(* CoDeSys 2.3 project: PRJ_LAB_AUTO_MAX4_V2200.pro *)
(* Title: Exam project *)
(* Version: 0.1 *)
(* Author: Federico M. Rossi *)
(* Description: Small project to take the exam.
Relased under MIT license. *)
(* Libraries: System_V002200.lib 3.4.06 14:28:36, PacDriveLib_V002002.lib 6.2.06 18:39:46 *)

(* Task configuration *)
TASK SymVisrtualAct (PRIORITY := 31, INTERVAL := T#100ms);
	SYM_PRG();
END_TASK
TASK Main (PRIORITY := 31, INTERVAL := T#10ms);
	PLC_PRG();
END_TASK

(* Global variable list: Global_Variables *)
VAR_GLOBAL
	tmpBool:BOOL;
	tmpReal:REAL;
	tmpDINT:DINT;
	tmpString:STRING(30);
	tmpTime:TIME;


	P1:virtual_piston_df_t;
	P2:virtual_piston_sfd_t;

	TP_PACK:BOOL:=FALSE;

	(* Machine config *)
	c:config_machine_t;




END_VAR

(* Data type *)
TYPE config_homing_t :
STRUCT
	maxTravel:REAL;
	vel:REAL;
	acc:REAL;
END_STRUCT
END_TYPE

(* Data type *)
TYPE config_machine_t :
STRUCT
	tape:config_tape_t;
	mov1:config_mov_t;
	mov2:config_mov_t;
	p1:config_piston_t;
	p2:config_piston_t;
	home1:config_homing_t;
	home2:config_homing_t;
END_STRUCT
END_TYPE

(* Data type *)
TYPE config_mov_t :
STRUCT
	acc:REAL;
	vel:REAL;
	pos:REAL;
	startForwAtTapePos:REAL;
	startBackAtTapePos:REAL;
END_STRUCT
END_TYPE

(* Data type *)
TYPE config_piston_t :
STRUCT
	deactAtTapePos:REAL;
END_STRUCT
END_TYPE

(* Data type *)
TYPE config_tape_t :
STRUCT
	acc:REAL;
	vel:REAL;
	period:REAL;
	packTimeoutSec:TIME;
END_STRUCT
END_TYPE

(* Data type *)
TYPE virtual_piston_df_i_t :
STRUCT
	setEnable:BOOL;
	setStart:BOOL;
END_STRUCT
END_TYPE

(* Data type *)
TYPE virtual_piston_df_o_t :
STRUCT
	isActive:BOOL;
	isOut:BOOL;
	isIn:BOOL;
END_STRUCT
END_TYPE

(* Data type *)
TYPE virtual_piston_df_t :
STRUCT
	i:virtual_piston_df_i_t;
	o:virtual_piston_df_o_t;
END_STRUCT
END_TYPE

(* Data type *)
TYPE virtual_piston_sfd_i_t :
STRUCT
	setEnable:BOOL;
	setStart:BOOL;
END_STRUCT
END_TYPE

(* Data type *)
TYPE virtual_piston_sfd_o_t :
STRUCT
	isActive:BOOL;
	isIn:BOOL;
END_STRUCT
END_TYPE

(* Data type *)
TYPE virtual_piston_sfd_t :
STRUCT
	i:virtual_piston_sfd_i_t;
	o:virtual_piston_sfd_o_t;
END_STRUCT
END_TYPE

(* POU SYM_PRG, ST *)
PROGRAM SYM_PRG
VAR

END_VAR
(* Piston 1 *)
IF ( P1.i.setEnable) THEN
	P1.o.isActive:=TRUE;
	IF ( P1.i.setStart) THEN
		p1.o.isIn:=FALSE;
		p1.o.isOut:=TRUE;
	ELSE
		p1.o.isIn:=TRUE;
		p1.o.isOut:=FALSE;
	END_IF
ELSE
	P1.o.isActive:=FALSE;
	P1.o.isIn:=FALSE;
	P1.o.isOut:=FALSE;
END_IF

(* Piston 2 *)
IF ( P2.i.setEnable) THEN
	P2.o.isActive:=TRUE;
	IF ( P2.i.setStart) THEN
		p2.o.isIn:=FALSE;
	ELSE
		p2.o.isIn:=TRUE;
	END_IF
ELSE
	P2.o.isActive:=FALSE;
	P2.o.isIn:=FALSE;
END_IF
END_PROGRAM

(* POU PLC_PRG, SFC *)
PROGRAM PLC_PRG
VAR
	exception:BOOL:=FALSE;

	(* axisMgmt => StateMachine *)
	enableOk:BOOL:=FALSE;
	homingOk:BOOL:=FALSE;
	syncStopOk:BOOL:=FALSE;
	tapeTimedOut:BOOL:=FALSE;
	(* StateMachine => axisMgmt *)
	AxisMgmtRoutine:INT:=0;

	(* tape related vars *)
	tape_pos_off:REAL;
	tape_pos_rel:REAL;
	flag_tp_pack:BOOL:=FALSE;
	timerTape:TON;
	jog1:Jogging3;
	jog2:Jogging3;
	elf_tape:EndlessFeed3;
	htp1:PDL_FB_HomeTP ;
	htp2:PDL_FB_HomeTP ;
	flagProcessingPack:BOOL;

	sm:STATE_MACHINE;
	OpModeReq:INT:=0;
	OpModeTimer:TON;
	stepReady:BOOL:=FALSE;
END_VAR
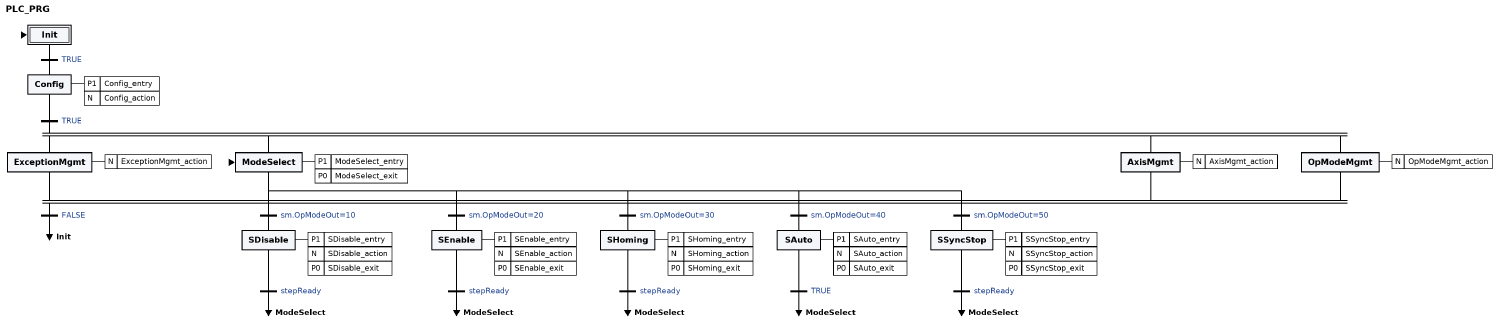
INITIAL_STEP Init:
END_STEP
TRANSITION FROM Init TO Config := TRUE;
END_TRANSITION
STEP Config:
	Config_entry(P1);
	Config_action(N);
END_STEP
TRANSITION FROM Config TO (ExceptionMgmt, ModeSelect, AxisMgmt, OpModeMgmt) := TRUE;
END_TRANSITION
STEP ExceptionMgmt:
	ExceptionMgmt_action(N);
END_STEP
STEP ModeSelect:
	ModeSelect_entry(P1);
	ModeSelect_exit(P0);
END_STEP
TRANSITION FROM ModeSelect TO SDisable := sm.OpModeOut=10;
END_TRANSITION
TRANSITION FROM ModeSelect TO SEnable := sm.OpModeOut=20;
END_TRANSITION
TRANSITION FROM ModeSelect TO SHoming := sm.OpModeOut=30;
END_TRANSITION
TRANSITION FROM ModeSelect TO SAuto := sm.OpModeOut=40;
END_TRANSITION
TRANSITION FROM ModeSelect TO SSyncStop := sm.OpModeOut=50;
END_TRANSITION
STEP SDisable:
	SDisable_entry(P1);
	SDisable_action(N);
	SDisable_exit(P0);
END_STEP
TRANSITION FROM SDisable TO ModeSelect := stepReady;
END_TRANSITION
STEP SEnable:
	SEnable_entry(P1);
	SEnable_action(N);
	SEnable_exit(P0);
END_STEP
TRANSITION FROM SEnable TO ModeSelect := stepReady;
END_TRANSITION
STEP SHoming:
	SHoming_entry(P1);
	SHoming_action(N);
	SHoming_exit(P0);
END_STEP
TRANSITION FROM SHoming TO ModeSelect := stepReady;
END_TRANSITION
STEP SAuto:
	SAuto_entry(P1);
	SAuto_action(N);
	SAuto_exit(P0);
END_STEP
TRANSITION FROM SAuto TO ModeSelect := TRUE;
END_TRANSITION
STEP SSyncStop:
	SSyncStop_entry(P1);
	SSyncStop_action(N);
	SSyncStop_exit(P0);
END_STEP
TRANSITION FROM SSyncStop TO ModeSelect := stepReady;
END_TRANSITION
STEP AxisMgmt:
	AxisMgmt_action(N);
END_STEP
STEP OpModeMgmt:
	OpModeMgmt_action(N);
END_STEP
TRANSITION FROM (ExceptionMgmt, AxisMgmt, OpModeMgmt) TO Init := FALSE;
END_TRANSITION

ACTION Config_entry:
	c.mov1.acc:=5000;
	c.mov1.pos:=90;
	c.mov1.startForwAtTapePos:=0;
	c.mov1.startBackAtTapePos:=180;
	c.mov1.vel:=90;

	c.mov2.acc:=5000;
	c.mov2.pos:=180;
	c.mov2.startForwAtTapePos:=360;
	c.mov2.startBackAtTapePos:=360+180;
	c.mov2.vel:=180;

	c.p1.deactAtTapePos:=180+45;
	c.p2.deactAtTapePos:=360+180+45;

	c.tape.acc:=5000;
	c.tape.packTimeoutSec:=t#30s;
	c.tape.period:=720;
	c.tape.vel:=72;

	c.home1.acc:=5000;
	c.home1.maxTravel:=750;
	c.home1.vel:=90;

	c.home2.acc:=5000;
	c.home2.maxTravel:=750;
	c.home2.vel:=90;
END_ACTION

ACTION Config_action:
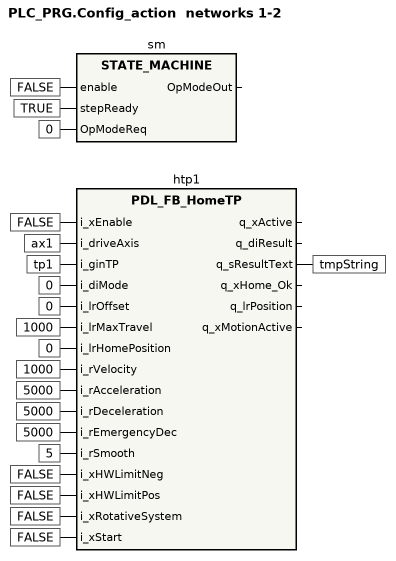
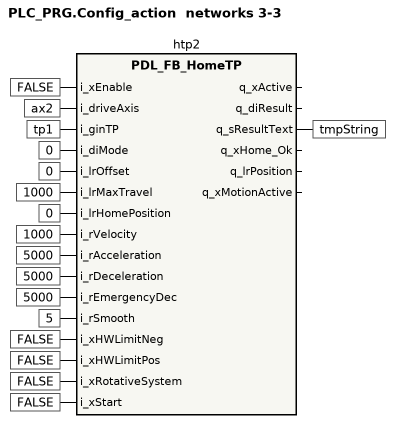
_FBD_ (* Function Block Diagram *)
NETWORK 1
	sm:STATE_MACHINE(enable: FALSE, stepReady: TRUE, OpModeReq: 0)
NETWORK 2
	htp1:PDL_FB_HomeTP(i_xEnable: FALSE, i_driveAxis: ax1, i_ginTP: tp1, i_diMode: 0, i_lrOffset: 0, i_lrMaxTravel: 1000, i_lrHomePosition: 0, i_rVelocity: 1000, i_rAcceleration: 5000, i_rDeceleration: 5000, i_rEmergencyDec: 5000, i_rSmooth: 5, i_xHWLimitNeg: FALSE, i_xHWLimitPos: FALSE, i_xRotativeSystem: FALSE, i_xStart: FALSE, q_sResultText => tmpString)
NETWORK 3
	htp2:PDL_FB_HomeTP(i_xEnable: FALSE, i_driveAxis: ax2, i_ginTP: tp1, i_diMode: 0, i_lrOffset: 0, i_lrMaxTravel: 1000, i_lrHomePosition: 0, i_rVelocity: 1000, i_rAcceleration: 5000, i_rDeceleration: 5000, i_rEmergencyDec: 5000, i_rSmooth: 5, i_xHWLimitNeg: FALSE, i_xHWLimitPos: FALSE, i_xRotativeSystem: FALSE, i_xStart: FALSE, q_sResultText => tmpString)
_END_FBD_
(* the same logic as Structured Text *)
(* Network 1 *)
sm(enable := FALSE, stepReady := TRUE, OpModeReq := 0);
(* Network 2 *)
htp1(i_xEnable := FALSE, i_driveAxis := ax1, i_ginTP := tp1, i_diMode := 0, i_lrOffset := 0, i_lrMaxTravel := 1000, i_lrHomePosition := 0, i_rVelocity := 1000, i_rAcceleration := 5000, i_rDeceleration := 5000, i_rEmergencyDec := 5000, i_rSmooth := 5, i_xHWLimitNeg := FALSE, i_xHWLimitPos := FALSE, i_xRotativeSystem := FALSE, i_xStart := FALSE);
tmpString := htp1.q_sResultText;
(* Network 3 *)
htp2(i_xEnable := FALSE, i_driveAxis := ax2, i_ginTP := tp1, i_diMode := 0, i_lrOffset := 0, i_lrMaxTravel := 1000, i_lrHomePosition := 0, i_rVelocity := 1000, i_rAcceleration := 5000, i_rDeceleration := 5000, i_rEmergencyDec := 5000, i_rSmooth := 5, i_xHWLimitNeg := FALSE, i_xHWLimitPos := FALSE, i_xRotativeSystem := FALSE, i_xStart := FALSE);
tmpString := htp2.q_sResultText;
END_ACTION

ACTION ExceptionMgmt_action:
(*
IF ( OpModeTimer.Q ) THEN
	exception:=TRUE;
END_IF
*)
IF (  exception ) THEN
	AxisMgmtRoutine:=0;
	stepReady:=TRUE;
	ax1.ControllerEnableSet:=FALSE;
	ax2.ControllerEnableSet:=FALSE;
	htp1.i_xEnable:=FALSE;
	htp2.i_xEnable:=FALSE;
	elf_tape.Enable:=FALSE;
	sm.enable:=FALSE;
END_IF
END_ACTION

ACTION ModeSelect_entry:
OpModeTimer.IN:=FALSE;
OpModeTimer.PT:=t#100s;
END_ACTION

ACTION ModeSelect_exit:
stepReady:=FALSE;
END_ACTION

ACTION SDisable_entry:
AxisMgmtRoutine:=10;
END_ACTION

ACTION SDisable_action:
IF ( (NOT enableOk) OR sm.OpModeOut<>10 ) THEN
	stepReady:=TRUE;
END_IF
END_ACTION

ACTION SDisable_exit:
AxisMgmtRoutine:=0;
END_ACTION

ACTION SEnable_entry:
AxisMgmtRoutine:=20;
OpModeTimer.PT:=t#10s;
OpModeTimer.IN:=TRUE;
END_ACTION

ACTION SEnable_action:
IF ( enableOk ) THEN
	stepReady:=TRUE;
END_IF
END_ACTION

ACTION SEnable_exit:
AxisMgmtRoutine:=0;
END_ACTION

ACTION SHoming_entry:
AxisMgmtRoutine:=30;
OpModeTimer.PT:=t#20s;
OpModeTimer.IN:=TRUE;
END_ACTION

ACTION SHoming_action:
IF ( homingOk ) THEN
	stepReady:=TRUE;
END_IF
END_ACTION

ACTION SHoming_exit:
AxisMgmtRoutine:=0;
END_ACTION

ACTION SAuto_entry:
OpModeTimer.IN:=FALSE;
END_ACTION

ACTION SAuto_action:
AxisMgmtRoutine:=40;
IF ( tapeTimedOut ) THEN
	OpModeReq:=50;
END_IF
END_ACTION

ACTION SAuto_exit:
AxisMgmtRoutine:=0;
END_ACTION

ACTION SSyncStop_entry:
OpModeTimer.IN:=FALSE;
END_ACTION

ACTION SSyncStop_action:
AxisMgmtRoutine:=50;
IF ( syncStopOk ) THEN
	stepReady:=TRUE;
END_IF
END_ACTION

ACTION SSyncStop_exit:
AxisMgmtRoutine:=0;
END_ACTION

ACTION AxisMgmt_action:
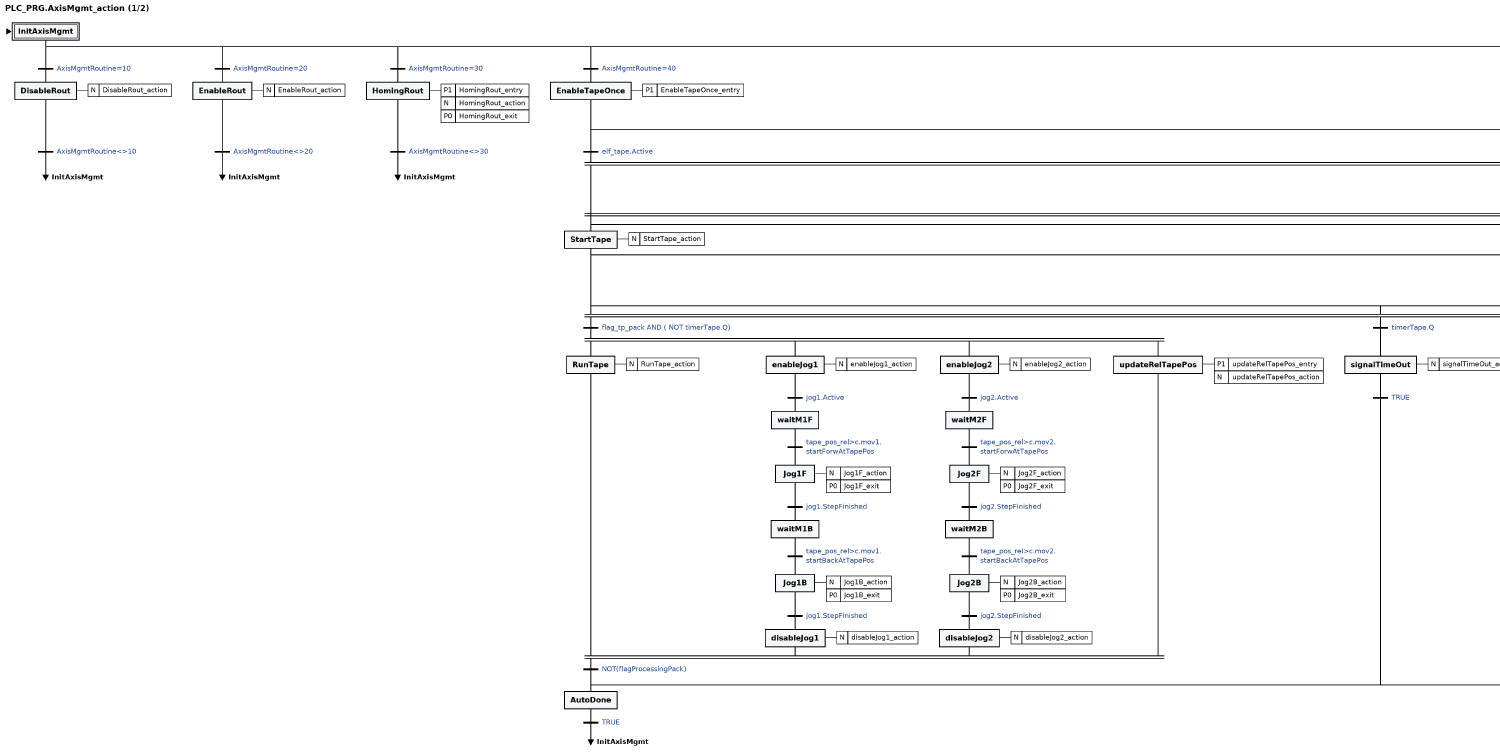
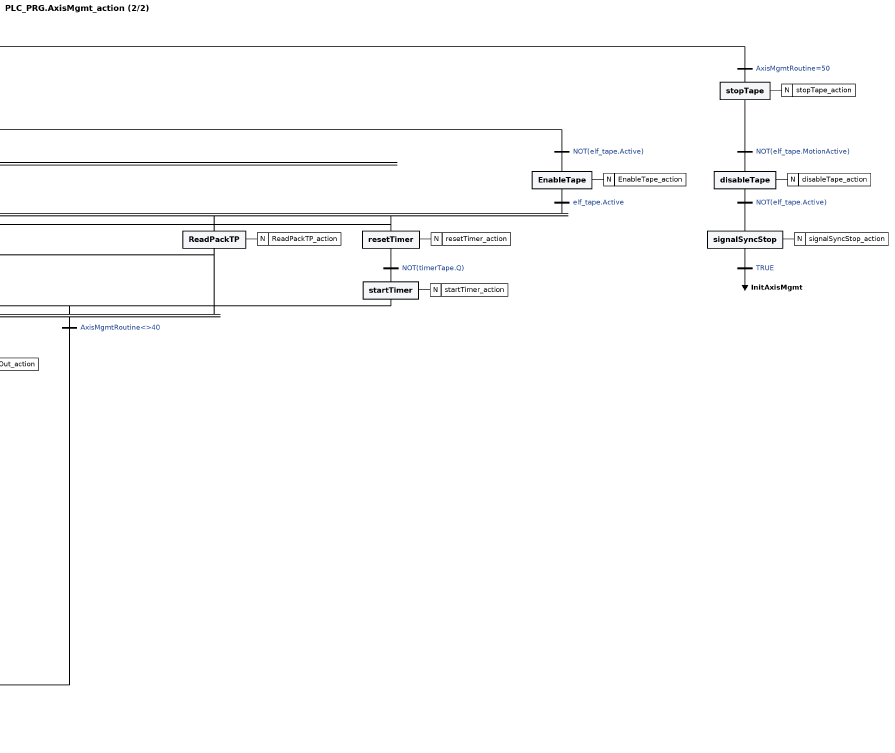
INITIAL_STEP InitAxisMgmt:
END_STEP
TRANSITION FROM InitAxisMgmt TO DisableRout := AxisMgmtRoutine=10;
END_TRANSITION
TRANSITION FROM InitAxisMgmt TO EnableRout := AxisMgmtRoutine=20;
END_TRANSITION
TRANSITION FROM InitAxisMgmt TO HomingRout := AxisMgmtRoutine=30;
END_TRANSITION
TRANSITION FROM InitAxisMgmt TO EnableTapeOnce := AxisMgmtRoutine=40;
END_TRANSITION
TRANSITION FROM InitAxisMgmt TO stopTape := AxisMgmtRoutine=50;
END_TRANSITION
STEP DisableRout:
	DisableRout_action(N);
END_STEP
TRANSITION FROM DisableRout TO InitAxisMgmt := AxisMgmtRoutine<>10;
END_TRANSITION
STEP EnableRout:
	EnableRout_action(N);
END_STEP
TRANSITION FROM EnableRout TO InitAxisMgmt := AxisMgmtRoutine<>20;
END_TRANSITION
STEP HomingRout:
	HomingRout_entry(P1);
	HomingRout_action(N);
	HomingRout_exit(P0);
END_STEP
TRANSITION FROM HomingRout TO InitAxisMgmt := AxisMgmtRoutine<>30;
END_TRANSITION
STEP EnableTapeOnce:
	EnableTapeOnce_entry(P1);
END_STEP
TRANSITION FROM EnableTapeOnce TO (StartTape, ReadPackTP, resetTimer) := elf_tape.Active;
END_TRANSITION
TRANSITION FROM EnableTapeOnce TO EnableTape := NOT(elf_tape.Active);
END_TRANSITION
STEP EnableTape:
	EnableTape_action(N);
END_STEP
TRANSITION FROM EnableTape TO (StartTape, ReadPackTP, resetTimer) := elf_tape.Active;
END_TRANSITION
STEP StartTape:
	StartTape_action(N);
END_STEP
STEP ReadPackTP:
	ReadPackTP_action(N);
END_STEP
STEP resetTimer:
	resetTimer_action(N);
END_STEP
TRANSITION FROM resetTimer TO startTimer := NOT(timerTape.Q);
END_TRANSITION
STEP startTimer:
	startTimer_action(N);
END_STEP
TRANSITION FROM (StartTape, ReadPackTP, startTimer) TO (RunTape, enableJog1, enableJog2, updateRelTapePos) := flag_tp_pack AND ( NOT timerTape.Q);
END_TRANSITION
TRANSITION FROM (StartTape, ReadPackTP, startTimer) TO signalTimeOut := timerTape.Q;
END_TRANSITION
TRANSITION FROM (StartTape, ReadPackTP, startTimer) TO AutoDone := AxisMgmtRoutine<>40;
END_TRANSITION
STEP RunTape:
	RunTape_action(N);
END_STEP
STEP enableJog1:
	enableJog1_action(N);
END_STEP
TRANSITION FROM enableJog1 TO waitM1F := jog1.Active;
END_TRANSITION
STEP waitM1F:
END_STEP
TRANSITION FROM waitM1F TO Jog1F := tape_pos_rel>c.mov1.startForwAtTapePos;
END_TRANSITION
STEP Jog1F:
	Jog1F_action(N);
	Jog1F_exit(P0);
END_STEP
TRANSITION FROM Jog1F TO waitM1B := jog1.StepFinished;
END_TRANSITION
STEP waitM1B:
END_STEP
TRANSITION FROM waitM1B TO Jog1B := tape_pos_rel>c.mov1.startBackAtTapePos;
END_TRANSITION
STEP Jog1B:
	Jog1B_action(N);
	Jog1B_exit(P0);
END_STEP
TRANSITION FROM Jog1B TO disableJog1 := jog1.StepFinished;
END_TRANSITION
STEP disableJog1:
	disableJog1_action(N);
END_STEP
STEP enableJog2:
	enableJog2_action(N);
END_STEP
TRANSITION FROM enableJog2 TO waitM2F := jog2.Active;
END_TRANSITION
STEP waitM2F:
END_STEP
TRANSITION FROM waitM2F TO Jog2F := tape_pos_rel>c.mov2.startForwAtTapePos;
END_TRANSITION
STEP Jog2F:
	Jog2F_action(N);
	Jog2F_exit(P0);
END_STEP
TRANSITION FROM Jog2F TO waitM2B := jog2.StepFinished;
END_TRANSITION
STEP waitM2B:
END_STEP
TRANSITION FROM waitM2B TO Jog2B := tape_pos_rel>c.mov2.startBackAtTapePos;
END_TRANSITION
STEP Jog2B:
	Jog2B_action(N);
	Jog2B_exit(P0);
END_STEP
TRANSITION FROM Jog2B TO disableJog2 := jog2.StepFinished;
END_TRANSITION
STEP disableJog2:
	disableJog2_action(N);
END_STEP
STEP updateRelTapePos:
	updateRelTapePos_entry(P1);
	updateRelTapePos_action(N);
END_STEP
TRANSITION FROM (RunTape, disableJog1, disableJog2, updateRelTapePos) TO AutoDone := NOT(flagProcessingPack);
END_TRANSITION
STEP signalTimeOut:
	signalTimeOut_action(N);
END_STEP
TRANSITION FROM signalTimeOut TO AutoDone := TRUE;
END_TRANSITION
STEP AutoDone:
END_STEP
TRANSITION FROM AutoDone TO InitAxisMgmt := TRUE;
END_TRANSITION
STEP stopTape:
	stopTape_action(N);
END_STEP
TRANSITION FROM stopTape TO disableTape := NOT(elf_tape.MotionActive);
END_TRANSITION
STEP disableTape:
	disableTape_action(N);
END_STEP
TRANSITION FROM disableTape TO signalSyncStop := NOT(elf_tape.Active);
END_TRANSITION
STEP signalSyncStop:
	signalSyncStop_action(N);
END_STEP
TRANSITION FROM signalSyncStop TO InitAxisMgmt := TRUE;
END_TRANSITION

ACTION DisableRout_action:
ax1.ControllerEnableSet := FALSE;
ax2.ControllerEnableSet := FALSE;
tape.ControllerEnableSet := FALSE;

IF ( ax1.AxisState=1 AND ax2.AxisState=1  ) THEN
	enableOk:=FALSE;
	homingOk:=FALSE;
	syncStopOk:=FALSE;
END_IF
END_ACTION

ACTION EnableRout_action:
ax1.ControllerEnableSet := TRUE;
ax2.ControllerEnableSet := TRUE;
tape.ControllerEnableSet := TRUE;

IF ( ax1.AxisState=3 AND ax2.AxisState=3 AND tape.AxisState=3) THEN
	enableOk:=TRUE;
	homingOk:=FALSE;
	syncStopOk:=FALSE;
ELSIF ( ax1.AxisState=8 OR ax2.AxisState=8 OR tape.AxisState=8  ) THEN
	exception:=TRUE;
END_IF
END_ACTION

ACTION HomingRout_entry:
htp1.i_xEnable:=TRUE;
htp2.i_xEnable:=TRUE;
homingOk:=FALSE;
syncStopOk:=FALSE;
END_ACTION

ACTION HomingRout_action:
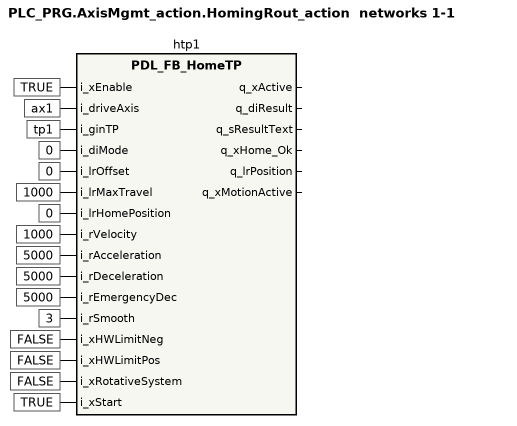
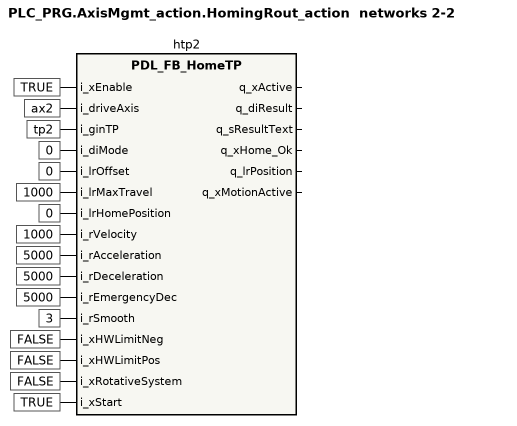
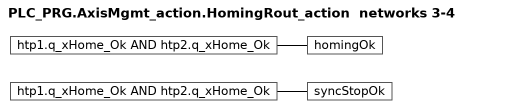
_FBD_ (* Function Block Diagram *)
NETWORK 1
	htp1:PDL_FB_HomeTP(i_xEnable: TRUE, i_driveAxis: ax1, i_ginTP: tp1, i_diMode: 0, i_lrOffset: 0, i_lrMaxTravel: 1000, i_lrHomePosition: 0, i_rVelocity: 1000, i_rAcceleration: 5000, i_rDeceleration: 5000, i_rEmergencyDec: 5000, i_rSmooth: 3, i_xHWLimitNeg: FALSE, i_xHWLimitPos: FALSE, i_xRotativeSystem: FALSE, i_xStart: TRUE)
NETWORK 2
	htp2:PDL_FB_HomeTP(i_xEnable: TRUE, i_driveAxis: ax2, i_ginTP: tp2, i_diMode: 0, i_lrOffset: 0, i_lrMaxTravel: 1000, i_lrHomePosition: 0, i_rVelocity: 1000, i_rAcceleration: 5000, i_rDeceleration: 5000, i_rEmergencyDec: 5000, i_rSmooth: 3, i_xHWLimitNeg: FALSE, i_xHWLimitPos: FALSE, i_xRotativeSystem: FALSE, i_xStart: TRUE)
NETWORK 3
	htp1.q_xHome_Ok AND htp2.q_xHome_Ok => homingOk
NETWORK 4
	htp1.q_xHome_Ok AND htp2.q_xHome_Ok => syncStopOk
_END_FBD_
(* the same logic as Structured Text *)
(* Network 1 *)
htp1(i_xEnable := TRUE, i_driveAxis := ax1, i_ginTP := tp1, i_diMode := 0, i_lrOffset := 0, i_lrMaxTravel := 1000, i_lrHomePosition := 0, i_rVelocity := 1000, i_rAcceleration := 5000, i_rDeceleration := 5000, i_rEmergencyDec := 5000, i_rSmooth := 3, i_xHWLimitNeg := FALSE, i_xHWLimitPos := FALSE, i_xRotativeSystem := FALSE, i_xStart := TRUE);
(* Network 2 *)
htp2(i_xEnable := TRUE, i_driveAxis := ax2, i_ginTP := tp2, i_diMode := 0, i_lrOffset := 0, i_lrMaxTravel := 1000, i_lrHomePosition := 0, i_rVelocity := 1000, i_rAcceleration := 5000, i_rDeceleration := 5000, i_rEmergencyDec := 5000, i_rSmooth := 3, i_xHWLimitNeg := FALSE, i_xHWLimitPos := FALSE, i_xRotativeSystem := FALSE, i_xStart := TRUE);
(* Network 3 *)
homingOk := htp1.q_xHome_Ok AND htp2.q_xHome_Ok;
(* Network 4 *)
syncStopOk := htp1.q_xHome_Ok AND htp2.q_xHome_Ok;
END_ACTION

ACTION HomingRout_exit:
htp1.i_xEnable:=FALSE;
htp2.i_xEnable:=FALSE;
END_ACTION

ACTION EnableTapeOnce_entry:
syncStopOk:=FALSE;
END_ACTION

ACTION EnableTape_action:
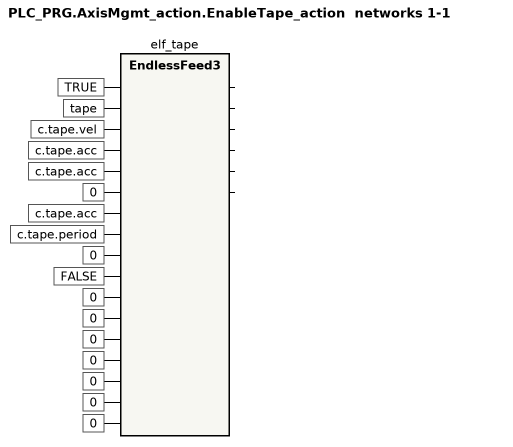
_FBD_ (* Function Block Diagram *)
NETWORK 1
	elf_tape:EndlessFeed3(TRUE, tape, c.tape.vel, c.tape.acc, c.tape.acc, 0, c.tape.acc, c.tape.period, 0, FALSE, 0, 0, 0, 0, 0, 0, 0)
_END_FBD_
(* the same logic as Structured Text *)
(* Network 1 *)
elf_tape(TRUE, tape, c.tape.vel, c.tape.acc, c.tape.acc, 0, c.tape.acc, c.tape.period, 0, FALSE, 0, 0, 0, 0, 0, 0, 0);
END_ACTION

ACTION StartTape_action:
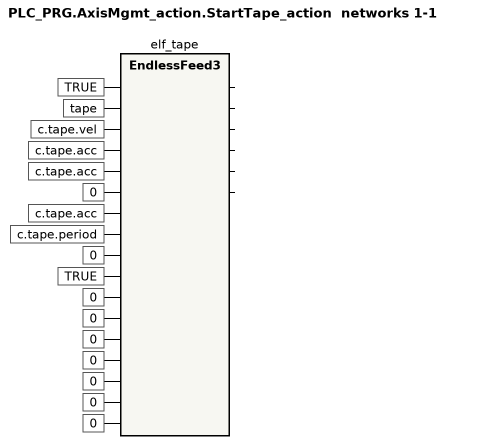
_FBD_ (* Function Block Diagram *)
NETWORK 1
	elf_tape:EndlessFeed3(TRUE, tape, c.tape.vel, c.tape.acc, c.tape.acc, 0, c.tape.acc, c.tape.period, 0, TRUE, 0, 0, 0, 0, 0, 0, 0)
_END_FBD_
(* the same logic as Structured Text *)
(* Network 1 *)
elf_tape(TRUE, tape, c.tape.vel, c.tape.acc, c.tape.acc, 0, c.tape.acc, c.tape.period, 0, TRUE, 0, 0, 0, 0, 0, 0, 0);
END_ACTION

ACTION ReadPackTP_action:
IF (  tp_PACK ) THEN
	IF ( NOT(flag_tp_pack) ) THEN
		flag_tp_pack:=TRUE;
		tape_pos_off:=tape.Position;
	END_IF
ELSE
	flag_tp_pack:=FALSE;
END_IF

(*
IF ( tape.Position > tape_pos_off ) THEN
	tape_pos_rel :=tape.Position -tape_pos_off;
ELSE
	tape_pos_rel :=tape.Position -tape_pos_off + c.tape.period;
END_IF
*)
tape_pos_rel:=0;
END_ACTION

ACTION resetTimer_action:
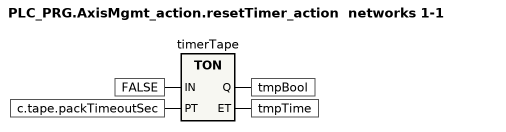
_FBD_ (* Function Block Diagram *)
NETWORK 1
	timerTape:TON(IN: FALSE, PT: c.tape.packTimeoutSec, ET => tmpTime) => tmpBool
_END_FBD_
(* the same logic as Structured Text *)
(* Network 1 *)
timerTape(IN := FALSE, PT := c.tape.packTimeoutSec);
tmpTime := timerTape.ET;
tmpBool := timerTape.Q;
END_ACTION

ACTION startTimer_action:
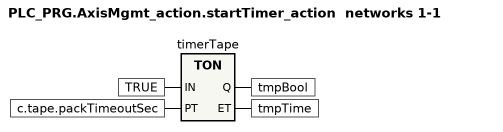
_FBD_ (* Function Block Diagram *)
NETWORK 1
	timerTape:TON(IN: TRUE, PT: c.tape.packTimeoutSec, ET => tmpTime) => tmpBool
_END_FBD_
(* the same logic as Structured Text *)
(* Network 1 *)
timerTape(IN := TRUE, PT := c.tape.packTimeoutSec);
tmpTime := timerTape.ET;
tmpBool := timerTape.Q;
END_ACTION

ACTION RunTape_action:
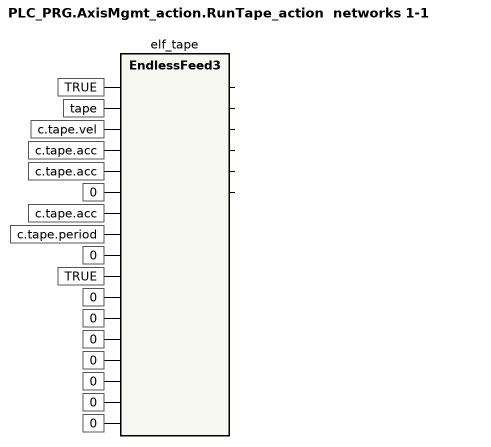
_FBD_ (* Function Block Diagram *)
NETWORK 1
	elf_tape:EndlessFeed3(TRUE, tape, c.tape.vel, c.tape.acc, c.tape.acc, 0, c.tape.acc, c.tape.period, 0, TRUE, 0, 0, 0, 0, 0, 0, 0)
_END_FBD_
(* the same logic as Structured Text *)
(* Network 1 *)
elf_tape(TRUE, tape, c.tape.vel, c.tape.acc, c.tape.acc, 0, c.tape.acc, c.tape.period, 0, TRUE, 0, 0, 0, 0, 0, 0, 0);
END_ACTION

ACTION enableJog1_action:
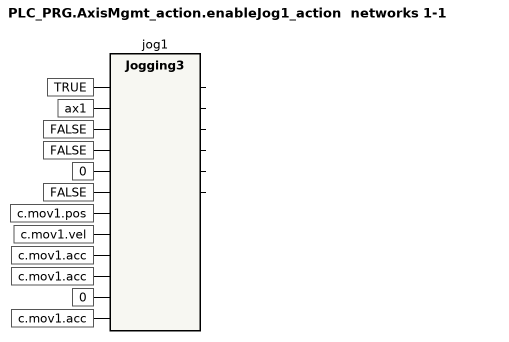
_FBD_ (* Function Block Diagram *)
NETWORK 1
	jog1:Jogging3(TRUE, ax1, FALSE, FALSE, 0, FALSE, c.mov1.pos, c.mov1.vel, c.mov1.acc, c.mov1.acc, 0, c.mov1.acc)
_END_FBD_
(* the same logic as Structured Text *)
(* Network 1 *)
jog1(TRUE, ax1, FALSE, FALSE, 0, FALSE, c.mov1.pos, c.mov1.vel, c.mov1.acc, c.mov1.acc, 0, c.mov1.acc);
END_ACTION

ACTION Jog1F_action:
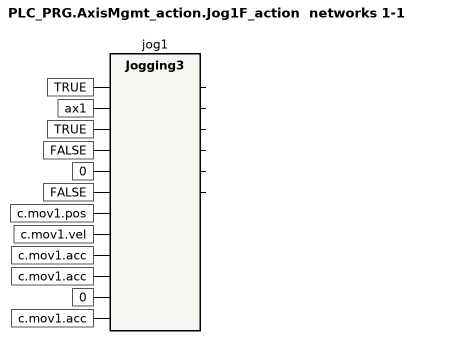
_FBD_ (* Function Block Diagram *)
NETWORK 1
	jog1:Jogging3(TRUE, ax1, TRUE, FALSE, 0, FALSE, c.mov1.pos, c.mov1.vel, c.mov1.acc, c.mov1.acc, 0, c.mov1.acc)
_END_FBD_
(* the same logic as Structured Text *)
(* Network 1 *)
jog1(TRUE, ax1, TRUE, FALSE, 0, FALSE, c.mov1.pos, c.mov1.vel, c.mov1.acc, c.mov1.acc, 0, c.mov1.acc);
END_ACTION

ACTION Jog1F_exit:
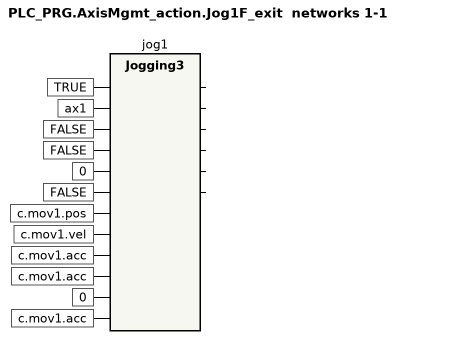
_FBD_ (* Function Block Diagram *)
NETWORK 1
	jog1:Jogging3(TRUE, ax1, FALSE, FALSE, 0, FALSE, c.mov1.pos, c.mov1.vel, c.mov1.acc, c.mov1.acc, 0, c.mov1.acc)
_END_FBD_
(* the same logic as Structured Text *)
(* Network 1 *)
jog1(TRUE, ax1, FALSE, FALSE, 0, FALSE, c.mov1.pos, c.mov1.vel, c.mov1.acc, c.mov1.acc, 0, c.mov1.acc);
END_ACTION

ACTION Jog1B_action:
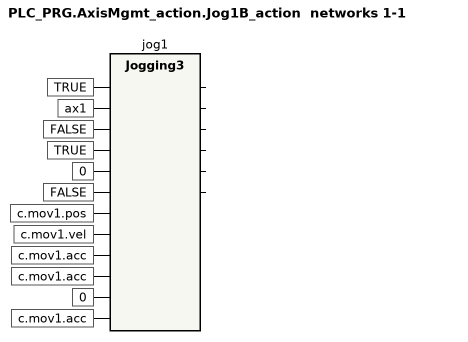
_FBD_ (* Function Block Diagram *)
NETWORK 1
	jog1:Jogging3(TRUE, ax1, FALSE, TRUE, 0, FALSE, c.mov1.pos, c.mov1.vel, c.mov1.acc, c.mov1.acc, 0, c.mov1.acc)
_END_FBD_
(* the same logic as Structured Text *)
(* Network 1 *)
jog1(TRUE, ax1, FALSE, TRUE, 0, FALSE, c.mov1.pos, c.mov1.vel, c.mov1.acc, c.mov1.acc, 0, c.mov1.acc);
END_ACTION

ACTION Jog1B_exit:
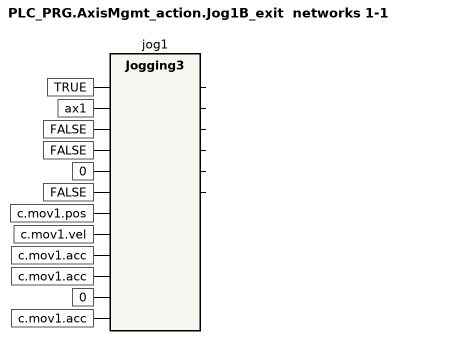
_FBD_ (* Function Block Diagram *)
NETWORK 1
	jog1:Jogging3(TRUE, ax1, FALSE, FALSE, 0, FALSE, c.mov1.pos, c.mov1.vel, c.mov1.acc, c.mov1.acc, 0, c.mov1.acc)
_END_FBD_
(* the same logic as Structured Text *)
(* Network 1 *)
jog1(TRUE, ax1, FALSE, FALSE, 0, FALSE, c.mov1.pos, c.mov1.vel, c.mov1.acc, c.mov1.acc, 0, c.mov1.acc);
END_ACTION

ACTION disableJog1_action:
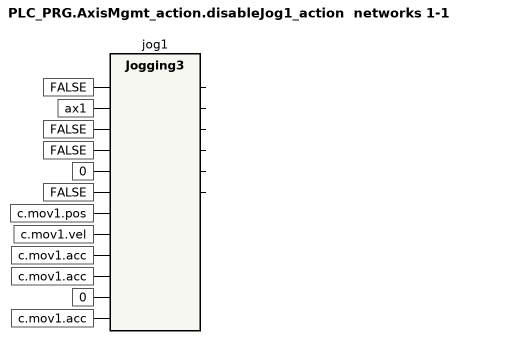
_FBD_ (* Function Block Diagram *)
NETWORK 1
	jog1:Jogging3(FALSE, ax1, FALSE, FALSE, 0, FALSE, c.mov1.pos, c.mov1.vel, c.mov1.acc, c.mov1.acc, 0, c.mov1.acc)
_END_FBD_
(* the same logic as Structured Text *)
(* Network 1 *)
jog1(FALSE, ax1, FALSE, FALSE, 0, FALSE, c.mov1.pos, c.mov1.vel, c.mov1.acc, c.mov1.acc, 0, c.mov1.acc);
END_ACTION

ACTION enableJog2_action:
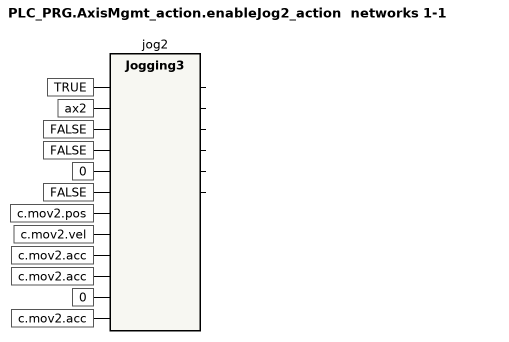
_FBD_ (* Function Block Diagram *)
NETWORK 1
	jog2:Jogging3(TRUE, ax2, FALSE, FALSE, 0, FALSE, c.mov2.pos, c.mov2.vel, c.mov2.acc, c.mov2.acc, 0, c.mov2.acc)
_END_FBD_
(* the same logic as Structured Text *)
(* Network 1 *)
jog2(TRUE, ax2, FALSE, FALSE, 0, FALSE, c.mov2.pos, c.mov2.vel, c.mov2.acc, c.mov2.acc, 0, c.mov2.acc);
END_ACTION

ACTION Jog2F_action:
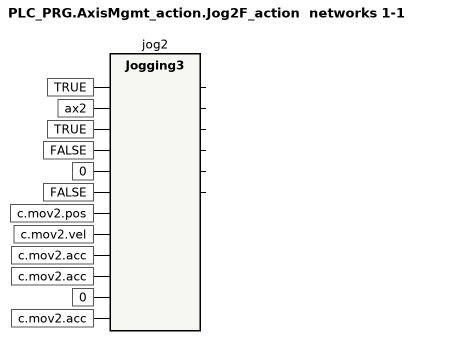
_FBD_ (* Function Block Diagram *)
NETWORK 1
	jog2:Jogging3(TRUE, ax2, TRUE, FALSE, 0, FALSE, c.mov2.pos, c.mov2.vel, c.mov2.acc, c.mov2.acc, 0, c.mov2.acc)
_END_FBD_
(* the same logic as Structured Text *)
(* Network 1 *)
jog2(TRUE, ax2, TRUE, FALSE, 0, FALSE, c.mov2.pos, c.mov2.vel, c.mov2.acc, c.mov2.acc, 0, c.mov2.acc);
END_ACTION

ACTION Jog2F_exit:
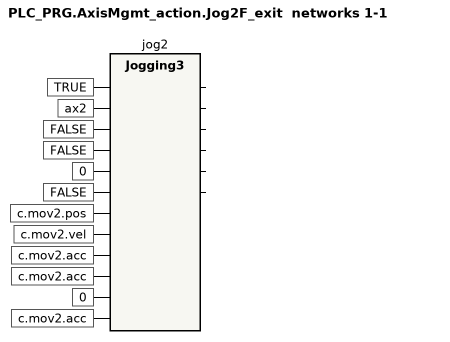
_FBD_ (* Function Block Diagram *)
NETWORK 1
	jog2:Jogging3(TRUE, ax2, FALSE, FALSE, 0, FALSE, c.mov2.pos, c.mov2.vel, c.mov2.acc, c.mov2.acc, 0, c.mov2.acc)
_END_FBD_
(* the same logic as Structured Text *)
(* Network 1 *)
jog2(TRUE, ax2, FALSE, FALSE, 0, FALSE, c.mov2.pos, c.mov2.vel, c.mov2.acc, c.mov2.acc, 0, c.mov2.acc);
END_ACTION

ACTION Jog2B_action:
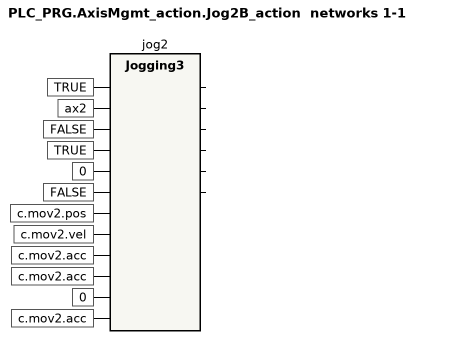
_FBD_ (* Function Block Diagram *)
NETWORK 1
	jog2:Jogging3(TRUE, ax2, FALSE, TRUE, 0, FALSE, c.mov2.pos, c.mov2.vel, c.mov2.acc, c.mov2.acc, 0, c.mov2.acc)
_END_FBD_
(* the same logic as Structured Text *)
(* Network 1 *)
jog2(TRUE, ax2, FALSE, TRUE, 0, FALSE, c.mov2.pos, c.mov2.vel, c.mov2.acc, c.mov2.acc, 0, c.mov2.acc);
END_ACTION

ACTION Jog2B_exit:
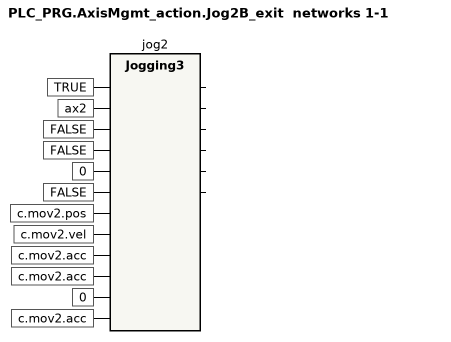
_FBD_ (* Function Block Diagram *)
NETWORK 1
	jog2:Jogging3(TRUE, ax2, FALSE, FALSE, 0, FALSE, c.mov2.pos, c.mov2.vel, c.mov2.acc, c.mov2.acc, 0, c.mov2.acc)
_END_FBD_
(* the same logic as Structured Text *)
(* Network 1 *)
jog2(TRUE, ax2, FALSE, FALSE, 0, FALSE, c.mov2.pos, c.mov2.vel, c.mov2.acc, c.mov2.acc, 0, c.mov2.acc);
END_ACTION

ACTION disableJog2_action:
